// TIA Portal V19 export
Screen "HOME PAGE"  NonexNone
